(* PLC project Generated.project, CODESYS CODESYS V3.5 SP19 Patch 1 *)
(* stored: creationDateTime 2026-08-18T12:52:51.295746, modificationDateTime 2026-08-18T12:52:51.295746 *)

(* ═══════════════════════════════════════════════════════════════ 🕹️ ST_JoystickHMI — Données d'échange IHM pour le Joystick ─────────────────────────────────────────────────────────────── 📄 Structuration en Cmd / State , homogène avec ST_ModesHMI. Pas de Cfg (les vrais réglages de calibration vivent dans GVL_PERSISTENT, pas ici) ni de Bypass (concept absent de ce struct). ═══════════════════════════════════════════════════════════════ *)
TYPE ST_JoystickHMI : STRUCT
  Cmd : ST_JoystickCmd;
  State : ST_JoystickState;
END_STRUCT;
END_TYPE

(* ═══════════════════════════════════════════════════════════════ 🎮 ST_JoystickCmd — Commandes IHM pour le Joystick ═══════════════════════════════════════════════════════════════ *)
TYPE ST_JoystickCmd : STRUCT
  BtnCalibrate : BOOL;  (* 🎯 Demande de recalage au neutre *)
END_STRUCT;
END_TYPE

(* ═══════════════════════════════════════════════════════════════ 🚦 ST_JoystickState — États et diagnostics IHM du Joystick ═══════════════════════════════════════════════════════════════ *)
TYPE ST_JoystickState : STRUCT
  RawX : INT;  (* 🕹️ Axe X brut du joystick (0..10000) *)
  RawY : INT;  (* 🕹️ Axe Y brut du joystick (0..10000) *)
  RawButton : BOOL;  (* 🔘 Bouton homme-mort brut *)
  AxisCmdX : ST_Joystick_AxisCmd;  (* ⚙️ Consigne d'axe X normalisée (sortie FB_Joystick) *)
  AxisCmdY : ST_Joystick_AxisCmd;  (* ⚙️ Consigne d'axe Y normalisée (sortie FB_Joystick) *)
  NeutralXAct : INT;  (* 🎯 Neutre X calibré actuel (lecture seule) *)
  NeutralYAct : INT;  (* 🎯 Neutre Y calibré actuel (lecture seule) *)
  DeadmanArmed : BOOL;  (* 🔫 Geste homme-mort armé (FB_Joystick.DeadmanArmed) *)
  AtNeutral : BOOL;  (* : TRUE si les 2 axes sont en zone morte (position centrale) *)
  Online : BOOL;  (* 📡 Liaison CAN joystick active *)
  Operational : BOOL;  (* 🟢 Joystick opérationnel *)
  Error : BOOL;  (* Joystick en défaut *)
  ErrorId : WORD;  (* ❌ Code défaut joystick *)
END_STRUCT;
END_TYPE

(* ======================================================================= 🕹️ ST_Joystick_AxisCmd — Consigne d'axe normalisée (sortie FB_Joystick) ─────────────────────────────────────────────────────────────── 🎯 Rôle : Structure de consigne d'axe 4 champs produite par FB_Joystick. 📤 Champs : Enable, StartStop, SpeedRef, Direction. 📄 Doc métier : DOC/AF/AF_Partie-08_Fonction_Joystick_v2.0.md ======================================================================= *)
TYPE ST_Joystick_AxisCmd : STRUCT
  Enable : BOOL;  (* === CONSIGNES DE PILOTAGE AXE === --> [CMD] Autorisation globale pipeline (FALSE=neutralisation, sorties coupees) *)
  StartStop : BOOL;  (* --> [CMD] Validation de mouvement (TRUE=acceleration, FALSE=deceleration) *)
  SpeedRef : REAL;  (* --> [CMD] Consigne vitesse signee (-100.0..+100.0 %, signe coherent avec Direction) *)
  Direction : INT;  (* --> [CMD] Sens de mouvement (-1=Arriere/Descente, 0=Neutre, +1=Avant/Montee) *)
END_STRUCT;
END_TYPE
